PROGRAM MAIN
VAR
END_VAR



	//备注测试

END_PROGRAM

(* stored: Version 1.1.0.1, ProductVersion 3.1.4024.9
   POU MAIN: Id {83f4e28e-4703-460b-98e7-32d6d206e679}, SpecialFunc None *)
